FUNCTION_BLOCK PUBLIC EventLoggerCaller
VAR_INPUT
END_VAR
VAR_OUTPUT
END_VAR
VAR_STAT
	test : TcMessage_Ext;
END_VAR

PROPERTY PUBLIC LoggerLevel : TcEventSeverity
GET
LoggerLevel := test.LoggerLevel;
END_GET
SET
test.LoggerLevel := LoggerLevel;
END_SET
END_PROPERTY

METHOD PUBLIC SendMessage : BOOL
VAR_INPUT
	eventType : Tc3_EventLogger.TcEventEntry;
	args : STRING(255);
END_VAR
test.Send(eventType := eventType, args := args);
END_METHOD

END_FUNCTION_BLOCK

(* stored: Version 1.1.0.1, ProductVersion 3.1.4024.11
   POU EventLoggerCaller: Id {3b332520-45e0-4fbd-8a12-5a5798153567}, SpecialFunc None
   Property LoggerLevel: Id {7a1da120-30ac-48b0-b143-72eb13841f05}
   Get Get: Id {d12ca7de-57d3-4365-b0d4-d095bb9a7ef4}
   Set Set: Id {07445f74-6004-4001-9016-db8d42ed9270}
   Method SendMessage: Id {27c653b0-052f-4876-8eb5-3aa962176d3e} *)
